FUNCTION_BLOCK fbInConveyor
VAR_INPUT
	SafetyOk			: BOOL;
	ResetCmd			: BOOL;
	AutoCycle			: BOOL;
	ManualCmd			: BOOL;
	
END_VAR
VAR_OUTPUT
	ResetCompleted 		: BOOL;
	
END_VAR
VAR
	FwdConveyor			AT %Q* :BOOL;
	State						: INT := 0;
END_VAR

END_FUNCTION_BLOCK

(* stored: Version 1.1.0.1, ProductVersion 3.1.4022.18
   POU fbInConveyor: Id {76ca436e-5ee1-43c3-bba6-80a39f7f3701}, SpecialFunc None *)
